// TIA Portal V19 export
FUNCTION "IFM_LMT100" : Void   // FC123, STL
TITLE = IFM_LMT100 IO_Link VendorID: 310 DeviceID:304
{ S7_Optimized_Access := 'TRUE' }
FAMILY : IO_Link
// stored: AutoNumber false
   VAR_INPUT
      Addr : Int;   // First Byte address of 4 byte address space
   END_VAR
   VAR_OUTPUT
      Level : Int;   // 2 bit offset, 14 bit integer, Current Level 0-100
      Out1 : Bool;
      Out2 : Bool;
   END_VAR
   VAR_TEMP
      TW_Flag : Word;
   END_VAR
BEGIN

NETWORK
TITLE = 
// Get first byte address
      L     #Addr;
      SLW   3;
      LAR1;

// 0-100% Current level
      L     IW [AR1, P#0.0];
      SRW   2;
      T     #Level;

//Output 1
      L     IB [AR1, P#0.0];
      T     #TW_Flag;
      L     1;
      AW;
      L     1;
      ==I;
      =     #Out1;

//Output 2
      L     IB [AR1, P#0.0];
      T     #TW_Flag;
      L     2;
      AW;
      L     2;
      ==I;
      =     #Out1;







END_FUNCTION
